PROGRAM main
VAR
	seg_a AT %QX0.0 : bool;
	seg_b AT %QX0.1 : bool;
	seg_c AT %QX0.2 : bool;
	seg_d AT %QX0.3 : bool;
	seg_e AT %QX0.4 : bool;
	seg_f AT %QX0.5 : bool;
	seg_g AT %QX0.6 : bool;
	BtnGreen AT %IX0.0 : bool;
	counter : int;
	seg1_display : Decoder7Seg;
	resetValue : int := 9;
	presetValue : int := 10;
	resetTrigger : bool;
	CTU1 : CTU;
	TON0 : TON;
	TON_Timer : time := T#30ms;
	TON_trigger : bool;
	Seg1_trigger : bool;
	CTU2 : CTU;
END_VAR

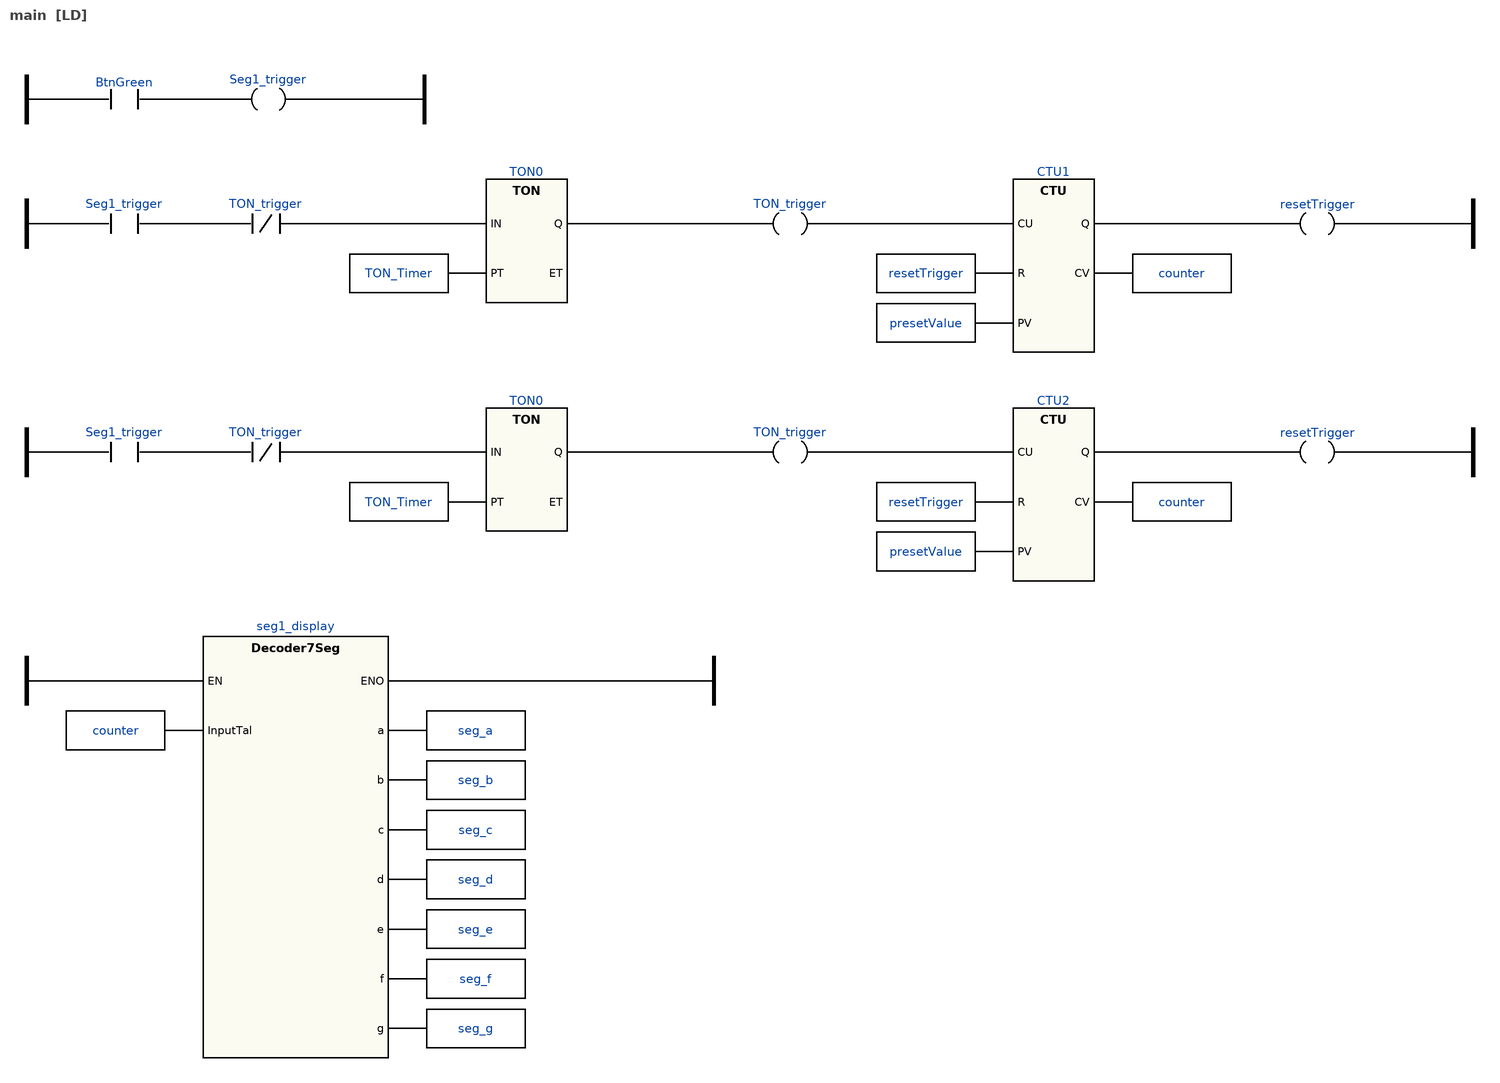
(* LD diagram, written out as Structured Text *)
Seg1_trigger := BtnGreen;
TON0(IN := Seg1_trigger AND NOT TON_trigger, PT := TON_Timer);
TON_trigger := TON0.Q;
CTU1(CU := TON0.Q, R := resetTrigger, PV := presetValue);
resetTrigger := CTU1.Q;
counter := CTU1.CV;
TON0(IN := Seg1_trigger AND NOT TON_trigger, PT := TON_Timer);
TON_trigger := TON0.Q;
CTU2(CU := TON0.Q, R := resetTrigger, PV := presetValue);
resetTrigger := CTU2.Q;
counter := CTU2.CV;
seg1_display(InputTal := counter);
seg_a := seg1_display.a;
seg_b := seg1_display.b;
seg_c := seg1_display.c;
seg_d := seg1_display.d;
seg_e := seg1_display.e;
seg_f := seg1_display.f;
seg_g := seg1_display.g;
END_PROGRAM
